// TIA Portal V15.1 export
// export: Created 2020-06-12T07:35:42.1318359Z, ExportSetting None, DisplayName Totally Integrated Automation Portal, DisplayVersion V15.1, DisplayName TIA Portal Openness, DisplayVersion V15.1, DisplayName STEP 7 Professional, DisplayVersion V15.1, DisplayName STEP 7 Safety, DisplayVersion V15.1, DisplayName WinCC Advanced, DisplayVersion V15.1
DATA_BLOCK "valid"   // DB26
{ S7_Optimized_Access := 'TRUE' }
AUTHOR : atec_osm
FAMILY : COMMON
NAME : AnaVal
VERSION : 2.0
// stored: MemoryReserve 100
   VAR
      ES1LD1_CV01 { ExternalAccessible := 'False'; ExternalVisible := 'False'; ExternalWritable := 'False'} : Bool := TRUE;   // Control Valve Dedusting System Position VALID
      ES1LV1_PT01 { ExternalAccessible := 'False'; ExternalVisible := 'False'; ExternalWritable := 'False'} : Bool := FALSE;   // Vacuum Pressure MPS FL VALID
      ES1LT1_XT01_volt { ExternalAccessible := 'False'; ExternalVisible := 'False'; ExternalWritable := 'False'} : Bool := TRUE;   // Actual voltage transducer VALID
      ES1LT1_XT01_pwr { ExternalAccessible := 'False'; ExternalVisible := 'False'; ExternalWritable := 'False'} : Bool := TRUE;   // Actual power transducer VALID
      ES1LT1_XT01_cur { ExternalAccessible := 'False'; ExternalVisible := 'False'; ExternalWritable := 'False'} : Bool := TRUE;   // Actual current transducer VALID
      ES1LT1_QT01 { ExternalAccessible := 'False'; ExternalVisible := 'False'; ExternalWritable := 'False'} : Bool := TRUE;   // Earth Leakage Current VALID
      ES1LV1_PT02 { ExternalAccessible := 'False'; ExternalVisible := 'False'; ExternalWritable := 'False'} : Bool := FALSE;   // Air Pressure MPS RL VALID
      ES1LT1_XS01_temp1 { ExternalAccessible := 'False'; ExternalVisible := 'False'; ExternalWritable := 'False'} : Bool := FALSE;   // Transformer Actual Temperature Coil U VALID
      ES1LT1_XS01_temp2 { ExternalAccessible := 'False'; ExternalVisible := 'False'; ExternalWritable := 'False'} : Bool := FALSE;   // Transformer Actual Temperature Coil V VALID
      ES1LT1_XS01_temp3 { ExternalAccessible := 'False'; ExternalVisible := 'False'; ExternalWritable := 'False'} : Bool := FALSE;   // Transformer Actual Temperature Coil W VALID
      ES1LA1_PT01 { ExternalAccessible := 'False'; ExternalVisible := 'False'; ExternalWritable := 'False'} : Bool := FALSE;   // Pressure Slag Bin VALID
      ES1LA2_PT01 { ExternalAccessible := 'False'; ExternalVisible := 'False'; ExternalWritable := 'False'} : Bool := TRUE;   // Pressure Sluice Alloy Addion VALID
      ES1LE2_M01pos { ExternalAccessible := 'False'; ExternalVisible := 'False'; ExternalWritable := 'False'} : Bool := TRUE;   // X-Adjustment Actual position VALID
      ES1LE2_M02pos { ExternalAccessible := 'False'; ExternalVisible := 'False'; ExternalWritable := 'False'} : Bool := TRUE;   // Y-Adjustment Actual position VALID
      ES1LC3_TT02 { ExternalAccessible := 'False'; ExternalVisible := 'False'; ExternalWritable := 'False'} : Bool := TRUE;   // Temperature Power Ram Outer Pipe RL VALID
      ES1LC3_TT04 { ExternalAccessible := 'False'; ExternalVisible := 'False'; ExternalWritable := 'False'} : Bool := TRUE;   // Temperature Conduction Rail 1+2 RL VALID
      ES1LC3_TT06 { ExternalAccessible := 'False'; ExternalVisible := 'False'; ExternalWritable := 'False'} : Bool := TRUE;   // Temperature Hood RL VALID
      ES1LE2_XT01 { ExternalAccessible := 'False'; ExternalVisible := 'False'; ExternalWritable := 'False'} : Bool := FALSE;   // Actual Voltage Power Ram VALID
      ES1LE3_PT01 { ExternalAccessible := 'False'; ExternalVisible := 'False'; ExternalWritable := 'False'} : Bool := FALSE;   // Pressure Protective Gas Hood 1 VALID
      ES1LE3_PT02 { ExternalAccessible := 'False'; ExternalVisible := 'False'; ExternalWritable := 'False'} : Bool := TRUE;   // Pressure Protective Gas Hood 2 VALID
      ES1LE3_QT01_O2 { ExternalAccessible := 'False'; ExternalVisible := 'False'; ExternalWritable := 'False'} : Bool := TRUE;   // Oxygen Measurement System VALID
      ES1LE3_QT01_O2hw { ExternalAccessible := 'False'; ExternalVisible := 'False'; ExternalWritable := 'False'} : Bool := FALSE;   // Oxygen Measurement System VALID
      ES1LE3_XT01 { ExternalAccessible := 'False'; ExternalVisible := 'False'; ExternalWritable := 'False'} : Bool := TRUE;   // Current Measuring Hood RL 1 act current VALID
      ES1LE3_XT02 { ExternalAccessible := 'False'; ExternalVisible := 'False'; ExternalWritable := 'False'} : Bool := TRUE;   // Current Measuring Hood RL 2 act current VALID
      ES1LE3_XT03 { ExternalAccessible := 'False'; ExternalVisible := 'False'; ExternalWritable := 'False'} : Bool := TRUE;   // Current Measuring Hood RL 3 act current VALID
      ES1LE3_XT04 { ExternalAccessible := 'False'; ExternalVisible := 'False'; ExternalWritable := 'False'} : Bool := TRUE;   // Current Measuring Hood RL 4 act current VALID
      ES1LZ1_PT01 { ExternalAccessible := 'False'; ExternalVisible := 'False'; ExternalWritable := 'False'} : Bool := TRUE;   // Pressure Atmosphere VALID
      ES1LC1_CV01 { ExternalAccessible := 'False'; ExternalVisible := 'False'; ExternalWritable := 'False'} : Bool := TRUE;   // Actual value Control valve RL Heat Exchanger VALID
      ES1LC1_PT01 { ExternalAccessible := 'False'; ExternalVisible := 'False'; ExternalWritable := 'False'} : Bool := TRUE;   // Foreward Line Strainer Pressure VALID
      ES1LC1_PT02 { ExternalAccessible := 'False'; ExternalVisible := 'False'; ExternalWritable := 'False'} : Bool := TRUE;   // Return Line Strainer Pressure VALID
      ES1LC1_dP02 { ExternalAccessible := 'False'; ExternalVisible := 'False'; ExternalWritable := 'False'} : Bool := FALSE;   // Differential pressure strainer VALID
      ES1LC1_PT03 { ExternalAccessible := 'False'; ExternalVisible := 'False'; ExternalWritable := 'False'} : Bool := TRUE;   // Pressure CW Tank VALID
      ES1LC1_QT01 { ExternalAccessible := 'False'; ExternalVisible := 'False'; ExternalWritable := 'False'} : Bool := TRUE;   // CW Tank actual conductivity VALID
      ES1LC1_TT01 { ExternalAccessible := 'False'; ExternalVisible := 'False'; ExternalWritable := 'False'} : Bool := TRUE;   // CW Tank Temperature VALID
      ES1LC1_TT02 { ExternalAccessible := 'False'; ExternalVisible := 'False'; ExternalWritable := 'False'} : Bool := TRUE;   // Temperature CW Recooling HE FL VALID
      ES1LC1_TT03 { ExternalAccessible := 'False'; ExternalVisible := 'False'; ExternalWritable := 'False'} : Bool := TRUE;   // Temperature CW Recooling HE RL VALID
      ES1LC1_TT04 { ExternalAccessible := 'False'; ExternalVisible := 'False'; ExternalWritable := 'False'} : Bool := TRUE;   // Temperature CW HE FL VALID
      ES1LC3_TT01 { ExternalAccessible := 'False'; ExternalVisible := 'False'; ExternalWritable := 'False'} : Bool := TRUE;   // Temperature Electrode Column RL VALID
      ES1LC5_CV01 { ExternalAccessible := 'False'; ExternalVisible := 'False'; ExternalWritable := 'False'} : Bool := TRUE;   // Control Valve CW MS1 Mould RL Position VALID
      ES1LC5_CV02 { ExternalAccessible := 'False'; ExternalVisible := 'False'; ExternalWritable := 'False'} : Bool := TRUE;   // Control Valve CW MS1 Baseplate RL Position VALID
      ES1LC5_FT01 { ExternalAccessible := 'False'; ExternalVisible := 'False'; ExternalWritable := 'False'} : Bool := TRUE;   // Flow CW Static Mould MS1 RL VALID
      ES1LC5_FT02 { ExternalAccessible := 'False'; ExternalVisible := 'False'; ExternalWritable := 'False'} : Bool := TRUE;   // Flow CW Baseplate MS1 RL VALID
      ES1LC5_PT01 { ExternalAccessible := 'False'; ExternalVisible := 'False'; ExternalWritable := 'False'} : Bool := TRUE;   // Pressure CW Melt Station 1 RL VALID
      ES1LC5_PT02 { ExternalAccessible := 'False'; ExternalVisible := 'False'; ExternalWritable := 'False'} : Bool := TRUE;   // Pressure CW Baseplate 1 RL value VALID
      ES1LC5_TT01 { ExternalAccessible := 'False'; ExternalVisible := 'False'; ExternalWritable := 'False'} : Bool := TRUE;   // Temperature CW Melt Station 1+2 FL VALID
      ES1LC5_TT02 { ExternalAccessible := 'False'; ExternalVisible := 'False'; ExternalWritable := 'False'} : Bool := TRUE;   // Temperature CW Static Mould MS1 RL VALID
      ES1LC5_TT04 { ExternalAccessible := 'False'; ExternalVisible := 'False'; ExternalWritable := 'False'} : Bool := TRUE;   // Temperature CW Baseplate 1 RL VALID
      ES1LC5_TT07 { ExternalAccessible := 'False'; ExternalVisible := 'False'; ExternalWritable := 'False'} : Bool := TRUE;   // Temperature Baseplate Clamp MS1 RL VALID
      ES1LC5_TT08 { ExternalAccessible := 'False'; ExternalVisible := 'False'; ExternalWritable := 'False'} : Bool := TRUE;   // Temperature Current Pipes MS1 RL VALID
      ES1LC6_CV01 { ExternalAccessible := 'False'; ExternalVisible := 'False'; ExternalWritable := 'False'} : Bool := TRUE;   // Control Valve CW MS2 Mould RL Position VALID
      ES1LC6_CV02 { ExternalAccessible := 'False'; ExternalVisible := 'False'; ExternalWritable := 'False'} : Bool := FALSE;   // Control Valve CW MS2 Baseplate RL Position VALID
      ES1LC6_FT01 { ExternalAccessible := 'False'; ExternalVisible := 'False'; ExternalWritable := 'False'} : Bool := TRUE;   // Flow CW Static Mould MS2 RL VALID
      ES1LC6_FT02 { ExternalAccessible := 'False'; ExternalVisible := 'False'; ExternalWritable := 'False'} : Bool := TRUE;   // Flow CW Baseplate 2 RL VALID
      ES1LC6_PT01 { ExternalAccessible := 'False'; ExternalVisible := 'False'; ExternalWritable := 'False'} : Bool := TRUE;   // Pressure CW Melt Station 2 RL VALID
      ES1LC6_PT02 { ExternalAccessible := 'False'; ExternalVisible := 'False'; ExternalWritable := 'False'} : Bool := TRUE;   // Pressure CW Baseplate 2 RL value VALID
      ES1LC6_TT02 { ExternalAccessible := 'False'; ExternalVisible := 'False'; ExternalWritable := 'False'} : Bool := TRUE;   // Temperature CW Static Mould MS2 RL VALID
      ES1LC6_TT04 { ExternalAccessible := 'False'; ExternalVisible := 'False'; ExternalWritable := 'False'} : Bool := TRUE;   // Temperature CW Baseplate 2 RL VALID
      ES1LC6_TT07 { ExternalAccessible := 'False'; ExternalVisible := 'False'; ExternalWritable := 'False'} : Bool := TRUE;   // Temperature Baseplate Clamp MS2 RL Actual value
      ES1LC6_TT08 { ExternalAccessible := 'False'; ExternalVisible := 'False'; ExternalWritable := 'False'} : Bool := TRUE;   // Temperature Current Pipes MS2 RL VALID
      ES1LC7_CV01 { ExternalAccessible := 'False'; ExternalVisible := 'False'; ExternalWritable := 'False'} : Bool := TRUE;   // Control Valve CW Module Recooling HE RL Position VALID
      ES1LC7_PT10 { ExternalAccessible := 'False'; ExternalVisible := 'False'; ExternalWritable := 'False'} : Bool := TRUE;   // Pressure CW Module Pump FL VALID
      ES1LC7_TT01 { ExternalAccessible := 'False'; ExternalVisible := 'False'; ExternalWritable := 'False'} : Bool := TRUE;   // Temperature CW Transductor RL VALID
      ES1LC7_TT02 { ExternalAccessible := 'False'; ExternalVisible := 'False'; ExternalWritable := 'False'} : Bool := TRUE;   // Temperature CW Current Condution F&amp;B RL VALID
      ES1LC7_TT10 { ExternalAccessible := 'False'; ExternalVisible := 'False'; ExternalWritable := 'False'} : Bool := TRUE;   // Temperature CW Module Pump FL VALID
      ES1LC7_TT12 { ExternalAccessible := 'False'; ExternalVisible := 'False'; ExternalWritable := 'False'} : Bool := TRUE;   // Temperature CW Module HE FL VALID
      ES1LC7_TT13 { ExternalAccessible := 'False'; ExternalVisible := 'False'; ExternalWritable := 'False'} : Bool := TRUE;   // Temperature CW Module HE RL VALID
      ES1LC7_TT14 { ExternalAccessible := 'False'; ExternalVisible := 'False'; ExternalWritable := 'False'} : Bool := TRUE;   // Temperature CW Module Recooling HE RL VALID
      ES1LC7_TT15 { ExternalAccessible := 'False'; ExternalVisible := 'False'; ExternalWritable := 'False'} : Bool := TRUE;   // Temperature CW Module Recooling HE FL VALID
      ES1LC7_TT16 { ExternalAccessible := 'False'; ExternalVisible := 'False'; ExternalWritable := 'False'} : Bool := TRUE;   // Temperature CW Vacuum Dry Screw Pump RL VALID
      ES1LC7_TT17 { ExternalAccessible := 'False'; ExternalVisible := 'False'; ExternalWritable := 'False'} : Bool := FALSE;   // Temperature CW Vacuum Roots Pump RL VALID
      ES1LC9_QT01 { ExternalAccessible := 'False'; ExternalVisible := 'False'; ExternalWritable := 'False'} : Bool := TRUE;
      ES1LC9_TT01 { ExternalAccessible := 'False'; ExternalVisible := 'False'; ExternalWritable := 'False'} : Bool := TRUE;
      ES1LC9_FT01 { ExternalAccessible := 'False'; ExternalVisible := 'False'; ExternalWritable := 'False'} : Bool := TRUE;
      ES1LC9_FT02 { ExternalAccessible := 'False'; ExternalVisible := 'False'; ExternalWritable := 'False'} : Bool := TRUE;
      ES1LC9_PT01 { ExternalAccessible := 'False'; ExternalVisible := 'False'; ExternalWritable := 'False'} : Bool := TRUE;
      ES1LG1_CV01 { ExternalAccessible := 'False'; ExternalVisible := 'False'; ExternalWritable := 'False'} : Bool := TRUE;   // Control Valve Ar PGH Act Flow VALID
      ES1LG1_CV02 { ExternalAccessible := 'False'; ExternalVisible := 'False'; ExternalWritable := 'False'} : Bool := FALSE;   // Control Valve N2 PGH Act Flow VALID
      ES1LA1_WT01 { ExternalAccessible := 'False'; ExternalVisible := 'False'; ExternalWritable := 'False'} : Bool := FALSE;   // Weight Slag Bin VALID
      ES1LA2_WT01 { ExternalAccessible := 'False'; ExternalVisible := 'False'; ExternalWritable := 'False'} : Bool := FALSE;   // Weight Alloy Bin VALID
      ES1LE1_WT01 { ExternalAccessible := 'False'; ExternalVisible := 'False'; ExternalWritable := 'False'} : Bool := FALSE;   // Weight Electrode Weight VALID
      AX1LD3_PT01 { ExternalAccessible := 'False'; ExternalVisible := 'False'; ExternalWritable := 'False'} : Bool := TRUE;   // Dedusting line pressure is valid
      AX1LD3_PT02 { ExternalAccessible := 'False'; ExternalVisible := 'False'; ExternalWritable := 'False'} : Bool := TRUE;   // Dedusting filter pressure is valid
   END_VAR
BEGIN
END_DATA_BLOCK
